(* IEC 61131-3 sources: esstee/src/tests/programs, 6 files *)

(* ---- arrays.ST ---- *)
VAR_GLOBAL
	arr1 : ARRAY [2..6] of INT;
	arr2 : ARRAY [-10..0] of INT;
	arr3 : ARRAY [0..1,0..2,0..3] of INT;
	arr4 : ARRAY [1..2,1..4,1..3] of INT :=
	     [
		[[1,2,3],[4,5,6],[7,8,9],[10,11,12]],
		[[21,22,23],[31,32,33],[34,35,36],[37,38,39]]
	     ];
END_VAR

PROGRAM t

;

END_PROGRAM

(* ---- conditionals.ST ---- *)
PROGRAM t_if

VAR
	i1 : DINT;
	i2 : DINT;
END_VAR

if i1 = 1 then
   i2 := 10;
elsif i1 = 2 then
   i2 := 20;
elsif i1 = 3 then
   i2 := 30;
else
   i2 := 40;
end_if;

END_PROGRAM

PROGRAM t_if_simple

VAR
	i1 : DINT;
	i2 : DINT := 20;
END_VAR

if i1 = 1 then
   i2 := 10;
end_if;

END_PROGRAM

PROGRAM t_case

VAR
	i1 : DINT;
	i2 : DINT;
END_VAR

case i1 of

1: i2 := 10;

2: i2 := 20;

3: i2 := 30;

else i2 := 40;

end_case;

END_PROGRAM

(* ---- directmemory.ST ---- *)
PROGRAM t

VAR
	b1 AT %MX0.0 : BOOL;
	b2 AT %MX0.1 : BOOL;
	b3 AT %MX0.2 : BOOL;
	b4 AT %MX0.3 : BOOL;
	b5 AT %MX0.4 : BOOL;
	b6 AT %MX0.5 : BOOL;
	b7 AT %MX0.6 : BOOL;
	b8 AT %MX0.7 : BOOL;

	b11 AT %MX1.0 : BOOL;
	b12 AT %MX1.1 : BOOL;
	b13 AT %MX1.2 : BOOL;
	b14 AT %MX1.3 : BOOL;
	b15 AT %MX1.4 : BOOL;
	b16 AT %MX1.5 : BOOL;
	b17 AT %MX1.6 : BOOL;
	b18 AT %MX1.7 : BOOL;

	s1 AT %MB0 : USINT;
	s2 AT %MB1 : USINT;
	s3 AT %MB2 : USINT;
	s4 AT %MB3 : USINT;
	s5 AT %MB4 : USINT;
	s6 AT %MB5 : USINT;
	s7 AT %MB6 : USINT;
	s8 AT %MB7 : USINT;

	i1 AT %MW0 : UINT;
	i2 AT %MW1 : UINT;
	i3 AT %MW2 : UINT;
	i4 AT %MW3 : UINT;

	d1 AT %MD0 : UDINT;
	d2 AT %MD1 : UDINT;

	l1 AT %ML0 : ULINT;
END_VAR

;

END_PROGRAM

(* ---- enum.ST ---- *)
VAR_GLOBAL
	e : (one, two, three);
	d : (single);
END_VAR

PROGRAM t

;

END_PROGRAM

(* ---- example.ST ---- *)
PROGRAM testprgm

VAR
	i: INT;
	a: UINT;
END_VAR

FOR i := 1 TO 20 DO

    IF i > 10 THEN
       a := 99;
    ELSE

        a := 10 - i;

    END_IF;

END_FOR;

END_PROGRAM

(* ---- literals.ST ---- *)
PROGRAM t

VAR
	i1 : DINT;
	i2 : DINT;
	i3 : DINT;
	i4 : DINT;

	t1 : TIME;

	r1 : REAL;
	r2 : REAL;

	b1 : BOOL;
	b2 : BOOL;

	td : TIME_OF_DAY;
	d1 : DATE;
	dd : DATE_AND_TIME;

	str : STRING;
	wstr : WSTRING;
END_VAR

;

END_PROGRAM

PROGRAM t_init

VAR
	i1 : DINT := 1;
	i2 : DINT := 2;
	i3 : DINT := 3;
	i4 : DINT := 4;

	t1 : TIME := T#1s;

	r1 : REAL := 1.0;
	r2 : REAL := 2.0;

	b1 : BOOL := true;
	b2 : BOOL := false;

	td : TIME_OF_DAY := TOD#10:10:10.10;
	d1 : DATE := D#1234-01-02;
	dd : DATE_AND_TIME := DT#1234-01-01-10:10:10.10;

	str : STRING := 'single';
	wstr : WSTRING := "double";
END_VAR

;

END_PROGRAM
